// TIA Portal V17 export
// export: Created 2024-06-14T09:53:09.4288461Z, ExportSetting WithDefaults, DisplayName Totally Integrated Automation Portal, DisplayVersion V17, DisplayName TIA Portal Openness, DisplayVersion V17, DisplayName TIA Portal Version Control Interface, DisplayVersion V17, DisplayName Simotion SCOUT TIA, DisplayVersion 5.4.3.0, DisplayName SINAMICS Startdrive Advanced, DisplayVersion V17 SP1 Update 1, DisplayName SINAMICS Startdrive G110M, G120, G120C, G120D, G120P, G115D, DisplayVersion V17 SP1 Update 1, DisplayName SINAMICS Startdrive G130, G150, S120, S150, SINAMICS MV, S210, DisplayVersion V17 SP1 Update 1, DisplayName STEP 7 Professional, DisplayVersion V17, DisplayName STEP 7 Safety, DisplayVersion V17, DisplayName WinCC Professional, DisplayVersion V17
FUNCTION_BLOCK "LPG_Check_scale_FB"   // FB102, LAD
TITLE = Fiiling Operation FB
{ S7_Optimized_Access := 'TRUE' }
VERSION : 0.1
// stored: AutoNumber false, IsIECCheckEnabled false, IsRetainMemResEnabled false, MemoryReserve 100, SetENOAutomatically false, UDAEnableTagReadback false
   VAR_INPUT
      INxCylinder_In_Pos : Bool;   // Cylinder In Position
      INxAuto_Start_Seq : Bool;   // Start Filling Sequence
      INxMan_Start_Seq : Bool;
      INxStop_Sequence : Bool;   // Stop Filling Sequence
      INtStart_TImeout_Time : DInt;   // Start Timeout Time in Sec
      INxReset_Sequence : Bool;   // Reset Sequence
      INxCylinder_Type : Int;
      INrTare_Entry_SP : Real;
      DOWN_CONVEYOR : Bool;
      data_delete : Bool;
   END_VAR
   VAR_OUTPUT
      OutuFilled_Data : Array[1..10] of Real;
      OutxDomestic_Cylinder : Bool;
      OutxCommercial_Cylinder : Bool;
      OutxStart_Timeout : Bool;
      OutxTare_Entry_Error : Bool;   // Coil 27
      Outx_Filling_Error : Bool;
      Outx_Tare_Value_Error : Bool;
      Cycle_Started : Bool;
      OutiStep_No : Int;
      OUTiResult : Int;
      Gross_Weight : Real;
      Net_Wieght : Real;
      Tare_Weight : Real;
      OUT_Decision : Int;
   END_VAR
   VAR_IN_OUT
      Modbus_Master_DB : "MOD_MASTER_DATA_1";
   END_VAR
   VAR
      TRIG : Array[1..25] of Bool;
      STEP_NO : Int;
      Step_Timer { S7_SetPoint := 'True'} : Array[1..15] of IEC_TIMER;
      Domestic_Cylinder { S7_SetPoint := 'True'} : Bool;
      Commercial_Cylinder : Bool;
      Cyl_Done { S7_SetPoint := 'True'} : TOF_TIME;
      Tare_Enrty_Extn { S7_SetPoint := 'True'} : TOF_TIME;
      Start_Timeout_Err { S7_SetPoint := 'True'} : TON_TIME;
      Tare_Entry_Timer { S7_SetPoint := 'True'} : TON_TIME;
      Filled_Gross : Real;
      Filled_Net : Real;
      Punched_Tare : Real;
      Test_Seq : Int;
      RESULT : Bool;
      IEC_Timer_0_Instance { S7_SetPoint := 'True'} : TOF_TIME;
      Gross { S7_SetPoint := 'True'} : Real;
      gross_diff : Real;
      pass : Bool;
      Decision : Word;
      IEC_Timer_0_Instance_1 { S7_SetPoint := 'True'} : TON_TIME;
      fill { S7_SetPoint := 'True'} : TON_TIME;
      ALL_FILL_DONE : Bool;
   END_VAR
   VAR RETAIN
      cycle_start { S7_SetPoint := 'True'} : CTU_INT;
   END_VAR
   VAR_TEMP
      Tare_Weight_Mul : Real;
      Tare_Enter_Time : DInt;
      Stt_TImeout_Time : DInt;
      Tare_Entry_Time : DInt;
      Tare_SP_Weigher : Int;
      Filled_Gross_Mul : Int;
      Filled_Net_Mul : Int;
      Filled_Tare_Mul : Int;
      "final wieght" : Real;
      final_weight_1 : Real;
   END_VAR
   // Tare_Enrty_Extn.PT := T#1s;
   VAR_TEMP   // added for the SCL form of the ladder/FBD networks
      _w1 : Bool;
      _w2 : Bool;
      _w3 : Bool;
   END_VAR
BEGIN

REGION Network 1: Empty Network
END_REGION

REGION Network 2: Input Mapping
END_REGION

REGION Network 3: Cylinder Selection ( Domestic / Commercial )
   // We have to receive from FIFO Entry-
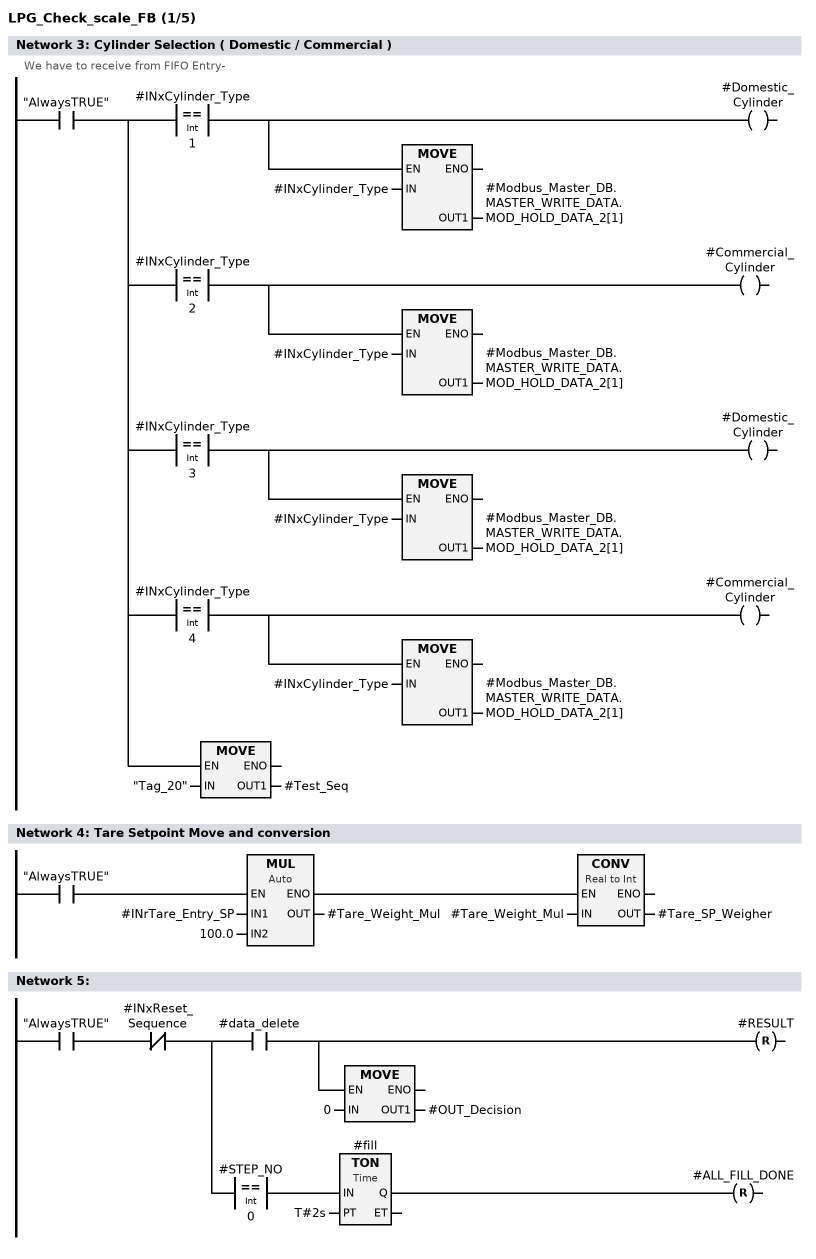
   RUNG wire#powerrail
      Contact( "AlwaysTRUE" )
      wire#w1
      { S7_Templates := "SrcType := Int" } EQ_Contact(in1 := #INxCylinder_Type, in2 := 1)
      wire#w2
      Coil( #Domestic_Cylinder )
   END_RUNG
   RUNG wire#w2
      Move(in := #INxCylinder_Type, out1 => #Modbus_Master_DB.MASTER_WRITE_DATA.MOD_HOLD_DATA_2[1])
   END_RUNG
   RUNG wire#w1
      { S7_Templates := "SrcType := Int" } EQ_Contact(in1 := #INxCylinder_Type, in2 := 2)
      wire#w3
      Coil( #Commercial_Cylinder )
   END_RUNG
   RUNG wire#w3
      Move(in := #INxCylinder_Type, out1 => #Modbus_Master_DB.MASTER_WRITE_DATA.MOD_HOLD_DATA_2[1])
   END_RUNG
   RUNG wire#w1
      { S7_Templates := "SrcType := Int" } EQ_Contact(in1 := #INxCylinder_Type, in2 := 3)
      wire#w4
      Coil( #Domestic_Cylinder )
   END_RUNG
   RUNG wire#w4
      Move(in := #INxCylinder_Type, out1 => #Modbus_Master_DB.MASTER_WRITE_DATA.MOD_HOLD_DATA_2[1])
   END_RUNG
   RUNG wire#w1
      { S7_Templates := "SrcType := Int" } EQ_Contact(in1 := #INxCylinder_Type, in2 := 4)
      wire#w5
      Coil( #Commercial_Cylinder )
   END_RUNG
   RUNG wire#w5
      Move(in := #INxCylinder_Type, out1 => #Modbus_Master_DB.MASTER_WRITE_DATA.MOD_HOLD_DATA_2[1])
   END_RUNG
   RUNG wire#w1
      Move(in := "Tag_20", out1 => #Test_Seq)
   END_RUNG
   // the same network as SCL:
   #Domestic_Cylinder := "AlwaysTRUE" AND (#INxCylinder_Type = 1);
   IF #Domestic_Cylinder THEN
       #Modbus_Master_DB.MASTER_WRITE_DATA.MOD_HOLD_DATA_2[1] := #INxCylinder_Type;
   END_IF;
   #Commercial_Cylinder := "AlwaysTRUE" AND (#INxCylinder_Type = 2);
   IF #Commercial_Cylinder THEN
       #Modbus_Master_DB.MASTER_WRITE_DATA.MOD_HOLD_DATA_2[1] := #INxCylinder_Type;
   END_IF;
   #Domestic_Cylinder := "AlwaysTRUE" AND (#INxCylinder_Type = 3);
   IF #Domestic_Cylinder THEN
       #Modbus_Master_DB.MASTER_WRITE_DATA.MOD_HOLD_DATA_2[1] := #INxCylinder_Type;
   END_IF;
   #Commercial_Cylinder := "AlwaysTRUE" AND (#INxCylinder_Type = 4);
   IF #Commercial_Cylinder THEN
       #Modbus_Master_DB.MASTER_WRITE_DATA.MOD_HOLD_DATA_2[1] := #INxCylinder_Type;
   END_IF;
   IF "AlwaysTRUE" THEN #Test_Seq := "Tag_20"; END_IF;
END_REGION

REGION Network 4: Tare Setpoint Move and conversion
   RUNG wire#powerrail
      Contact( "AlwaysTRUE" )
      Mul(in1 := #INrTare_Entry_SP, in2 := 100.0, out => #Tare_Weight_Mul)
      { S7_Templates := "[SrcType := Real, DestType := Int]" } Convert(in := #Tare_Weight_Mul, out => #Tare_SP_Weigher)
   END_RUNG
   // the same network as SCL:
   IF "AlwaysTRUE" THEN
       #Tare_Weight_Mul := #INrTare_Entry_SP * 100.0;
       #Tare_SP_Weigher := REAL_TO_INT(#Tare_Weight_Mul);
   END_IF;
END_REGION

REGION Network 5
   RUNG wire#powerrail
      Contact( "AlwaysTRUE" )
      I_Contact( #INxReset_Sequence )
      wire#w1
      Contact( #data_delete )
      wire#w2
      R_Coil( #RESULT )
   END_RUNG
   RUNG wire#w2
      Move(in := 0, out1 => #OUT_Decision)
   END_RUNG
   RUNG wire#w1
      { S7_Templates := "SrcType := Int" } EQ_Contact(in1 := #STEP_NO, in2 := 0)
      { S7_Templates := "time_type := Time" } #fill.TON(pt := T#2s, et =>)
      R_Coil( #ALL_FILL_DONE )
   END_RUNG
   // the same network as SCL:
   #_w1 := "AlwaysTRUE" AND NOT #INxReset_Sequence;
   IF #_w1 AND #data_delete THEN
       #RESULT := FALSE;
       #OUT_Decision := 0;
   END_IF;
   #fill(IN := #_w1 AND (#STEP_NO = 0), PT := T#2s);   // TON
   IF #fill.Q THEN #ALL_FILL_DONE := FALSE; END_IF;
END_REGION

REGION Network 6: Cylinder Selection
   // Cylinder Selection will write the logic later
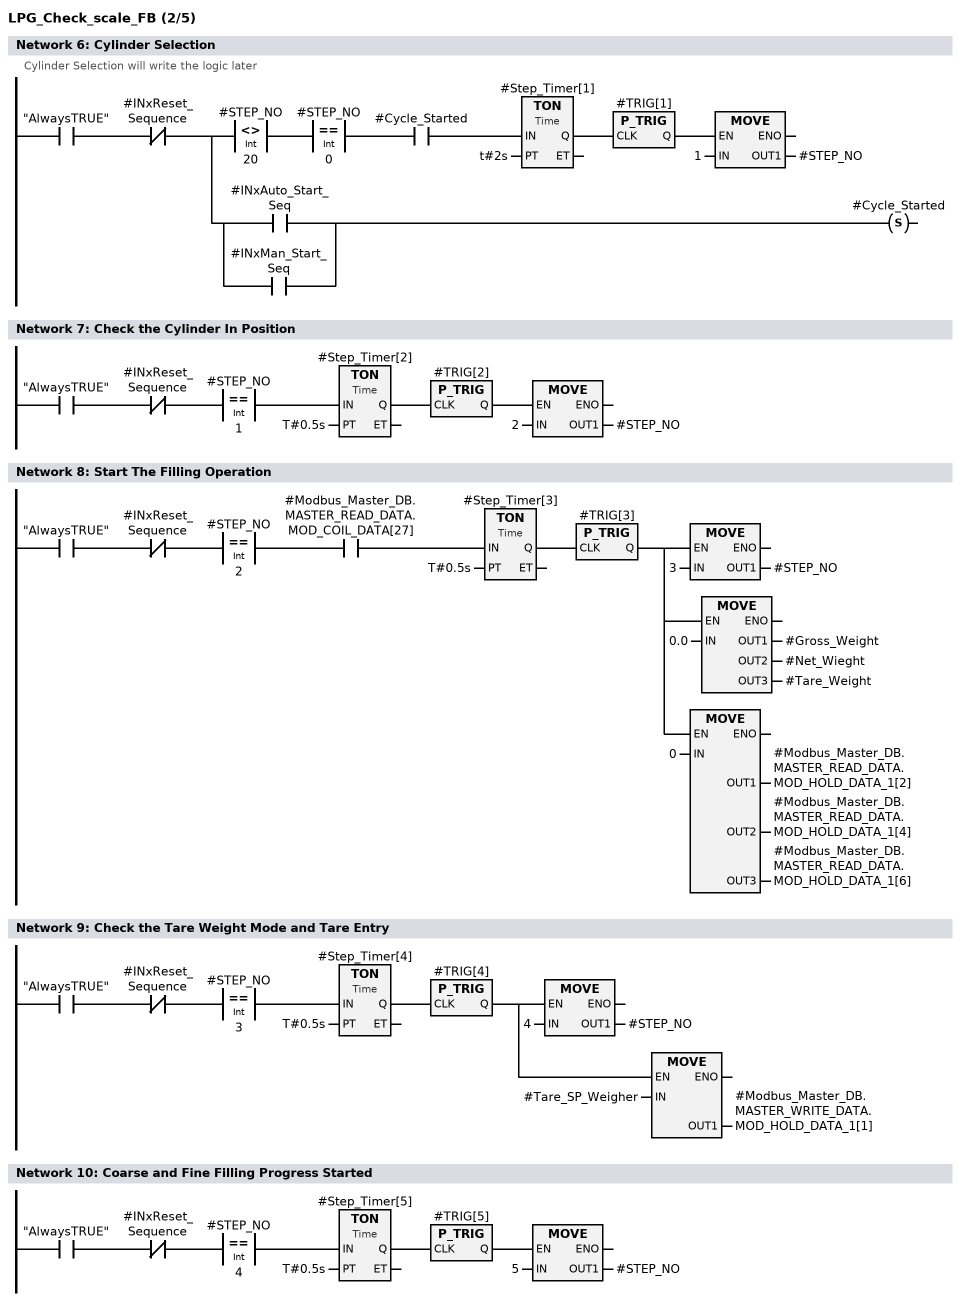
   RUNG wire#powerrail
      Contact( "AlwaysTRUE" )
      I_Contact( #INxReset_Sequence )
      wire#w1
      { S7_Templates := "SrcType := Int" } NE_Contact(in1 := #STEP_NO, in2 := 20)
      { S7_Templates := "SrcType := Int" } EQ_Contact(in1 := #STEP_NO, in2 := 0)
      Contact( #Cycle_Started )
      { S7_Templates := "time_type := Time" } #Step_Timer[1].TON(pt := t#2s, et =>)
      P_Trig( #TRIG[1] )
      Move(in := 1, out1 => #STEP_NO)
   END_RUNG
   RUNG wire#w1
      Contact( #INxAuto_Start_Seq )
      wire#w2
      S_Coil( #Cycle_Started )
   END_RUNG
   RUNG wire#w1
      Contact( #INxMan_Start_Seq )
   END_RUNG wire#w2
   // the same network as SCL:
   #_w1 := "AlwaysTRUE" AND NOT #INxReset_Sequence;
   #Step_Timer[1].TON(IN := #_w1 AND (#STEP_NO <> 20) AND (#STEP_NO = 0) AND #Cycle_Started, PT := t#2s);
   #_w2 := #Step_Timer[1].Q AND NOT #TRIG[1];   // rising edge
   #TRIG[1] := #Step_Timer[1].Q;
   IF #_w2 THEN #STEP_NO := 1; END_IF;
   IF #_w1 AND (#INxAuto_Start_Seq OR #INxMan_Start_Seq) THEN #Cycle_Started := TRUE; END_IF;
END_REGION

REGION Network 7: Check the Cylinder In Position
   RUNG wire#powerrail
      Contact( "AlwaysTRUE" )
      I_Contact( #INxReset_Sequence )
      { S7_Templates := "SrcType := Int" } EQ_Contact(in1 := #STEP_NO, in2 := 1)
      { S7_Templates := "time_type := Time" } #Step_Timer[2].TON(pt := T#0.5s, et =>)
      P_Trig( #TRIG[2] )
      Move(in := 2, out1 => #STEP_NO)
   END_RUNG
   // the same network as SCL:
   #Step_Timer[2].TON(IN := "AlwaysTRUE" AND NOT #INxReset_Sequence AND (#STEP_NO = 1), PT := T#0.5s);
   #_w1 := #Step_Timer[2].Q AND NOT #TRIG[2];   // rising edge
   #TRIG[2] := #Step_Timer[2].Q;
   IF #_w1 THEN #STEP_NO := 2; END_IF;
END_REGION

REGION Network 8: Start The Filling Operation
   RUNG wire#powerrail
      Contact( "AlwaysTRUE" )
      I_Contact( #INxReset_Sequence )
      { S7_Templates := "SrcType := Int" } EQ_Contact(in1 := #STEP_NO, in2 := 2)
      Contact( #Modbus_Master_DB.MASTER_READ_DATA.MOD_COIL_DATA[27] )
      { S7_Templates := "time_type := Time" } #Step_Timer[3].TON(pt := T#0.5s, et =>)
      P_Trig( #TRIG[3] )
      wire#w1
      Move(in := 3, out1 => #STEP_NO)
   END_RUNG
   RUNG wire#w1
      Move(in := 0.0, out1 => #Gross_Weight, out2 => #Net_Wieght, out3 => #Tare_Weight)
   END_RUNG
   RUNG wire#w1
      Move(in := 0, out1 => #Modbus_Master_DB.MASTER_READ_DATA.MOD_HOLD_DATA_1[2], out2 => #Modbus_Master_DB.MASTER_READ_DATA.MOD_HOLD_DATA_1[4], out3 => #Modbus_Master_DB.MASTER_READ_DATA.MOD_HOLD_DATA_1[6])
   END_RUNG
   // the same network as SCL:
   #Step_Timer[3].TON(IN := "AlwaysTRUE" AND NOT #INxReset_Sequence AND (#STEP_NO = 2) AND #Modbus_Master_DB.MASTER_READ_DATA.MOD_COIL_DATA[27],
                      PT := T#0.5s);
   #_w1 := #Step_Timer[3].Q AND NOT #TRIG[3];   // rising edge
   #TRIG[3] := #Step_Timer[3].Q;
   IF #_w1 THEN
       #STEP_NO := 3;
       #Gross_Weight := 0.0;
       #Net_Wieght := 0.0;
       #Tare_Weight := 0.0;
       #Modbus_Master_DB.MASTER_READ_DATA.MOD_HOLD_DATA_1[2] := 0;
       #Modbus_Master_DB.MASTER_READ_DATA.MOD_HOLD_DATA_1[4] := 0;
       #Modbus_Master_DB.MASTER_READ_DATA.MOD_HOLD_DATA_1[6] := 0;
   END_IF;
END_REGION

REGION Network 9: Check the Tare Weight Mode and Tare Entry
   RUNG wire#powerrail
      Contact( "AlwaysTRUE" )
      I_Contact( #INxReset_Sequence )
      { S7_Templates := "SrcType := Int" } EQ_Contact(in1 := #STEP_NO, in2 := 3)
      { S7_Templates := "time_type := Time" } #Step_Timer[4].TON(pt := T#0.5s, et =>)
      P_Trig( #TRIG[4] )
      wire#w1
      Move(in := 4, out1 => #STEP_NO)
   END_RUNG
   RUNG wire#w1
      Move(in := #Tare_SP_Weigher, out1 => #Modbus_Master_DB.MASTER_WRITE_DATA.MOD_HOLD_DATA_1[1])
   END_RUNG
   // the same network as SCL:
   #Step_Timer[4].TON(IN := "AlwaysTRUE" AND NOT #INxReset_Sequence AND (#STEP_NO = 3), PT := T#0.5s);
   #_w1 := #Step_Timer[4].Q AND NOT #TRIG[4];   // rising edge
   #TRIG[4] := #Step_Timer[4].Q;
   IF #_w1 THEN
       #STEP_NO := 4;
       #Modbus_Master_DB.MASTER_WRITE_DATA.MOD_HOLD_DATA_1[1] := #Tare_SP_Weigher;
   END_IF;
END_REGION

REGION Network 10: Coarse and Fine Filling Progress Started
   RUNG wire#powerrail
      Contact( "AlwaysTRUE" )
      I_Contact( #INxReset_Sequence )
      { S7_Templates := "SrcType := Int" } EQ_Contact(in1 := #STEP_NO, in2 := 4)
      { S7_Templates := "time_type := Time" } #Step_Timer[5].TON(pt := T#0.5s, et =>)
      P_Trig( #TRIG[5] )
      Move(in := 5, out1 => #STEP_NO)
   END_RUNG
   // the same network as SCL:
   #Step_Timer[5].TON(IN := "AlwaysTRUE" AND NOT #INxReset_Sequence AND (#STEP_NO = 4), PT := T#0.5s);
   #_w1 := #Step_Timer[5].Q AND NOT #TRIG[5];   // rising edge
   #TRIG[5] := #Step_Timer[5].Q;
   IF #_w1 THEN #STEP_NO := 5; END_IF;
END_REGION

REGION Network 11: Coarse Filling Completed
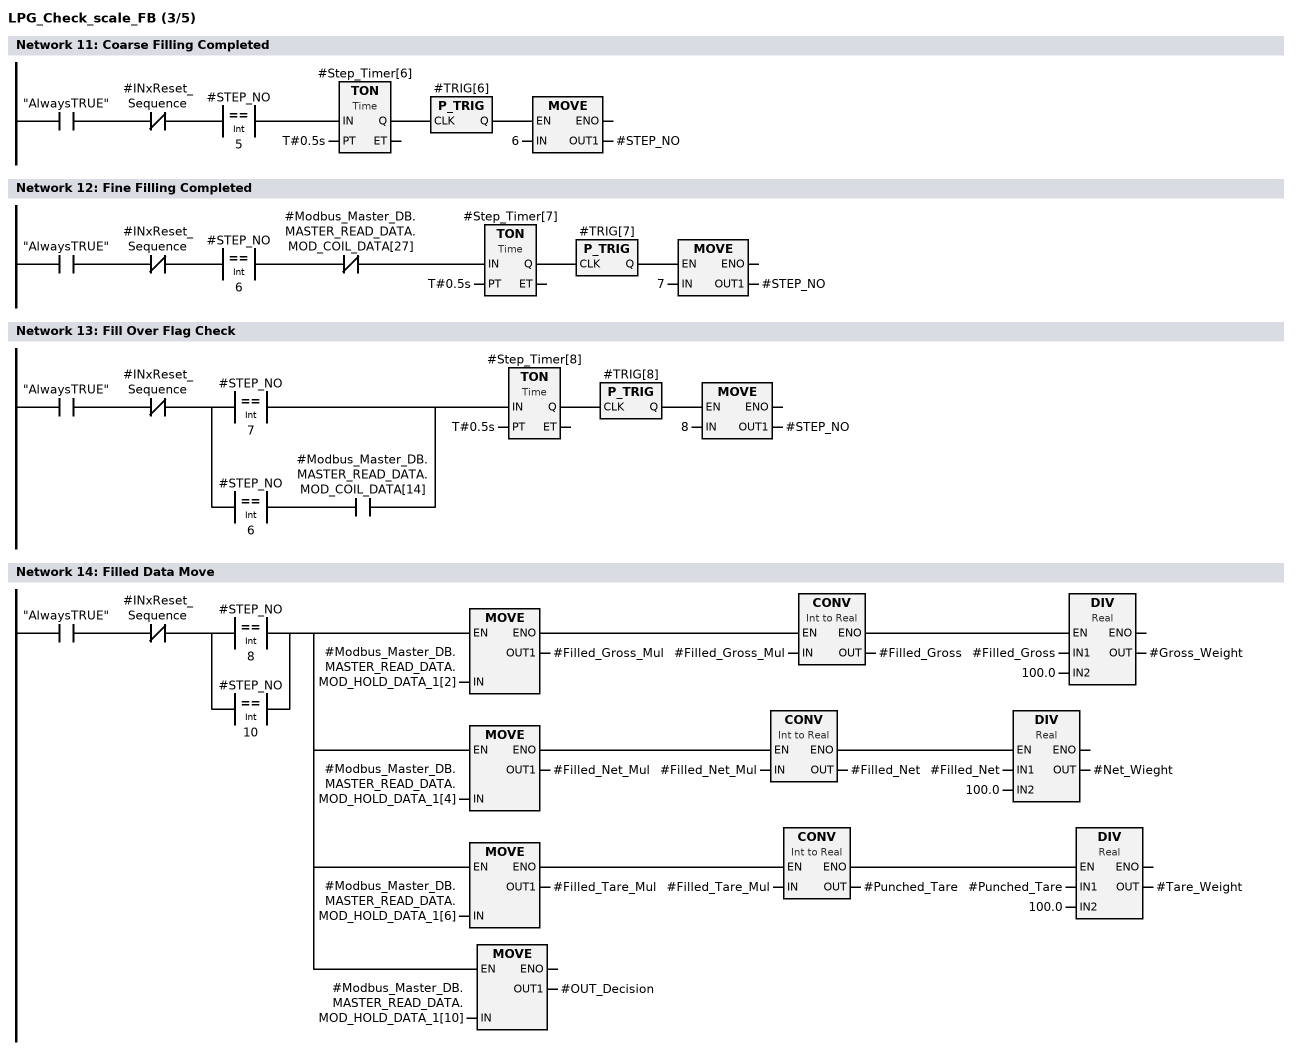
   RUNG wire#powerrail
      Contact( "AlwaysTRUE" )
      I_Contact( #INxReset_Sequence )
      { S7_Templates := "SrcType := Int" } EQ_Contact(in1 := #STEP_NO, in2 := 5)
      { S7_Templates := "time_type := Time" } #Step_Timer[6].TON(pt := T#0.5s, et =>)
      P_Trig( #TRIG[6] )
      Move(in := 6, out1 => #STEP_NO)
   END_RUNG
   // the same network as SCL:
   #Step_Timer[6].TON(IN := "AlwaysTRUE" AND NOT #INxReset_Sequence AND (#STEP_NO = 5), PT := T#0.5s);
   #_w1 := #Step_Timer[6].Q AND NOT #TRIG[6];   // rising edge
   #TRIG[6] := #Step_Timer[6].Q;
   IF #_w1 THEN #STEP_NO := 6; END_IF;
END_REGION

REGION Network 12: Fine Filling Completed
   RUNG wire#powerrail
      Contact( "AlwaysTRUE" )
      I_Contact( #INxReset_Sequence )
      { S7_Templates := "SrcType := Int" } EQ_Contact(in1 := #STEP_NO, in2 := 6)
      I_Contact( #Modbus_Master_DB.MASTER_READ_DATA.MOD_COIL_DATA[27] )
      { S7_Templates := "time_type := Time" } #Step_Timer[7].TON(pt := T#0.5s, et =>)
      P_Trig( #TRIG[7] )
      Move(in := 7, out1 => #STEP_NO)
   END_RUNG
   // the same network as SCL:
   #Step_Timer[7].TON(IN := "AlwaysTRUE" AND NOT #INxReset_Sequence AND (#STEP_NO = 6) AND NOT #Modbus_Master_DB.MASTER_READ_DATA.MOD_COIL_DATA[27],
                      PT := T#0.5s);
   #_w1 := #Step_Timer[7].Q AND NOT #TRIG[7];   // rising edge
   #TRIG[7] := #Step_Timer[7].Q;
   IF #_w1 THEN #STEP_NO := 7; END_IF;
END_REGION

REGION Network 13: Fill Over Flag Check
   RUNG wire#powerrail
      Contact( "AlwaysTRUE" )
      I_Contact( #INxReset_Sequence )
      wire#w1
      { S7_Templates := "SrcType := Int" } EQ_Contact(in1 := #STEP_NO, in2 := 7)
      wire#w2
      { S7_Templates := "time_type := Time" } #Step_Timer[8].TON(pt := T#0.5s, et =>)
      P_Trig( #TRIG[8] )
      Move(in := 8, out1 => #STEP_NO)
   END_RUNG
   RUNG wire#w1
      { S7_Templates := "SrcType := Int" } EQ_Contact(in1 := #STEP_NO, in2 := 6)
      Contact( #Modbus_Master_DB.MASTER_READ_DATA.MOD_COIL_DATA[14] )
   END_RUNG wire#w2
   // the same network as SCL:
   #Step_Timer[8].TON(IN := "AlwaysTRUE" AND NOT #INxReset_Sequence AND ((#STEP_NO = 7) OR ((#STEP_NO = 6) AND #Modbus_Master_DB.MASTER_READ_DATA.MOD_COIL_DATA[14])),
                      PT := T#0.5s);
   #_w1 := #Step_Timer[8].Q AND NOT #TRIG[8];   // rising edge
   #TRIG[8] := #Step_Timer[8].Q;
   IF #_w1 THEN #STEP_NO := 8; END_IF;
END_REGION

REGION Network 14: Filled Data Move
   RUNG wire#powerrail
      Contact( "AlwaysTRUE" )
      I_Contact( #INxReset_Sequence )
      wire#w1
      { S7_Templates := "SrcType := Int" } EQ_Contact(in1 := #STEP_NO, in2 := 8)
      wire#w2
      Move(in := #Modbus_Master_DB.MASTER_READ_DATA.MOD_HOLD_DATA_1[2], out1 => #Filled_Gross_Mul)
      { S7_Templates := "[SrcType := Int, DestType := Real]" } Convert(in := #Filled_Gross_Mul, out => #Filled_Gross)
      { S7_Templates := "SrcType := Real" } Div(in1 := #Filled_Gross, in2 := 100.0, out => #Gross_Weight)
   END_RUNG
   RUNG wire#w1
      { S7_Templates := "SrcType := Int" } EQ_Contact(in1 := #STEP_NO, in2 := 10)
   END_RUNG wire#w2
   RUNG wire#w2
      Move(in := #Modbus_Master_DB.MASTER_READ_DATA.MOD_HOLD_DATA_1[4], out1 => #Filled_Net_Mul)
      { S7_Templates := "[SrcType := Int, DestType := Real]" } Convert(in := #Filled_Net_Mul, out => #Filled_Net)
      { S7_Templates := "SrcType := Real" } Div(in1 := #Filled_Net, in2 := 100.0, out => #Net_Wieght)
   END_RUNG
   RUNG wire#w2
      Move(in := #Modbus_Master_DB.MASTER_READ_DATA.MOD_HOLD_DATA_1[6], out1 => #Filled_Tare_Mul)
      { S7_Templates := "[SrcType := Int, DestType := Real]" } Convert(in := #Filled_Tare_Mul, out => #Punched_Tare)
      { S7_Templates := "SrcType := Real" } Div(in1 := #Punched_Tare, in2 := 100.0, out => #Tare_Weight)
   END_RUNG
   RUNG wire#w2
      Move(in := #Modbus_Master_DB.MASTER_READ_DATA.MOD_HOLD_DATA_1[10], out1 => #OUT_Decision)
   END_RUNG
   // the same network as SCL:
   IF "AlwaysTRUE" AND NOT #INxReset_Sequence AND ((#STEP_NO = 8) OR (#STEP_NO = 10)) THEN
       #Filled_Gross_Mul := #Modbus_Master_DB.MASTER_READ_DATA.MOD_HOLD_DATA_1[2];
       #Filled_Gross := INT_TO_REAL(#Filled_Gross_Mul);
       #Gross_Weight := #Filled_Gross / 100.0;
       #Filled_Net_Mul := #Modbus_Master_DB.MASTER_READ_DATA.MOD_HOLD_DATA_1[4];
       #Filled_Net := INT_TO_REAL(#Filled_Net_Mul);
       #Net_Wieght := #Filled_Net / 100.0;
       #Filled_Tare_Mul := #Modbus_Master_DB.MASTER_READ_DATA.MOD_HOLD_DATA_1[6];
       #Punched_Tare := INT_TO_REAL(#Filled_Tare_Mul);
       #Tare_Weight := #Punched_Tare / 100.0;
       #OUT_Decision := #Modbus_Master_DB.MASTER_READ_DATA.MOD_HOLD_DATA_1[10];
   END_IF;
END_REGION

REGION Network 15: Filling Operation Complete
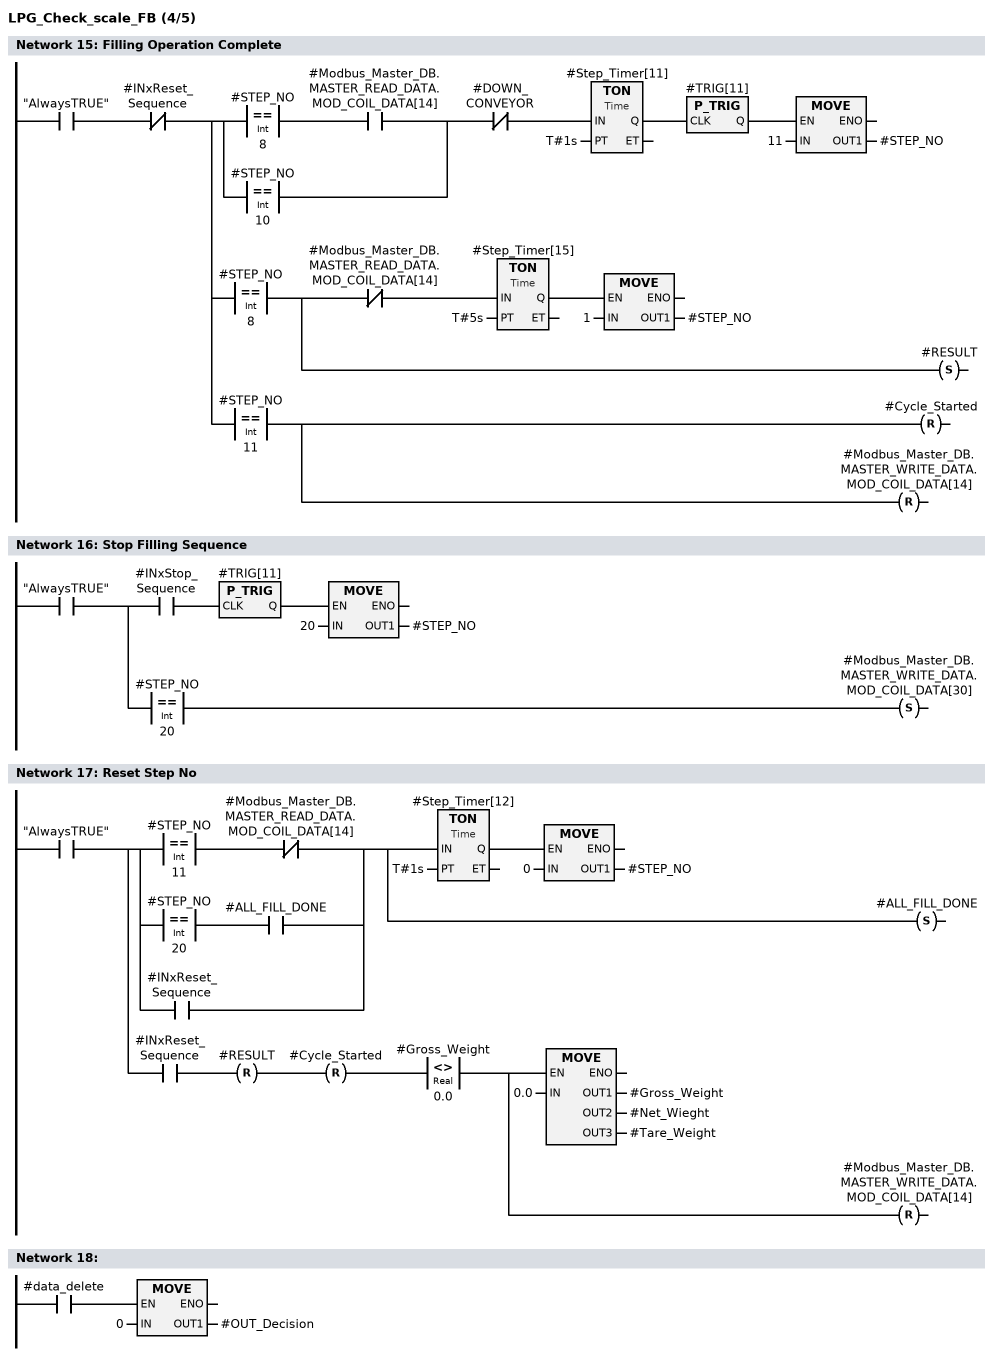
   RUNG wire#powerrail
      Contact( "AlwaysTRUE" )
      I_Contact( #INxReset_Sequence )
      wire#w1
      { S7_Templates := "SrcType := Int" } EQ_Contact(in1 := #STEP_NO, in2 := 8)
      Contact( #Modbus_Master_DB.MASTER_READ_DATA.MOD_COIL_DATA[14] )
      wire#w2
      I_Contact( #DOWN_CONVEYOR )
      { S7_Templates := "time_type := Time" } #Step_Timer[11].TON(pt := T#1s, et =>)
      P_Trig( #TRIG[11] )
      Move(in := 11, out1 => #STEP_NO)
   END_RUNG
   RUNG wire#w1
      { S7_Templates := "SrcType := Int" } EQ_Contact(in1 := #STEP_NO, in2 := 10)
   END_RUNG wire#w2
   RUNG wire#w1
      { S7_Templates := "SrcType := Int" } EQ_Contact(in1 := #STEP_NO, in2 := 8)
      wire#w3
      I_Contact( #Modbus_Master_DB.MASTER_READ_DATA.MOD_COIL_DATA[14] )
      { S7_Templates := "time_type := Time" } #Step_Timer[15].TON(pt := T#5s, et =>)
      Move(in := 1, out1 => #STEP_NO)
   END_RUNG
   RUNG wire#w3
      S_Coil( #RESULT )
   END_RUNG
   RUNG wire#w1
      { S7_Templates := "SrcType := Int" } EQ_Contact(in1 := #STEP_NO, in2 := 11)
      wire#w4
      R_Coil( #Cycle_Started )
   END_RUNG
   RUNG wire#w4
      R_Coil( #Modbus_Master_DB.MASTER_WRITE_DATA.MOD_COIL_DATA[14] )
   END_RUNG
   // the same network as SCL:
   #_w1 := "AlwaysTRUE" AND NOT #INxReset_Sequence;
   #Step_Timer[11].TON(IN := #_w1 AND (((#STEP_NO = 8) AND #Modbus_Master_DB.MASTER_READ_DATA.MOD_COIL_DATA[14]) OR (#STEP_NO = 10)) AND NOT #DOWN_CONVEYOR,
                       PT := T#1s);
   #_w2 := #Step_Timer[11].Q AND NOT #TRIG[11];   // rising edge
   #TRIG[11] := #Step_Timer[11].Q;
   IF #_w2 THEN #STEP_NO := 11; END_IF;
   #_w3 := #_w1 AND (#STEP_NO = 8);
   #Step_Timer[15].TON(IN := #_w3 AND NOT #Modbus_Master_DB.MASTER_READ_DATA.MOD_COIL_DATA[14], PT := T#5s);
   IF #Step_Timer[15].Q THEN #STEP_NO := 1; END_IF;
   IF #_w3 THEN #RESULT := TRUE; END_IF;
   IF #_w1 AND (#STEP_NO = 11) THEN
       #Cycle_Started := FALSE;
       #Modbus_Master_DB.MASTER_WRITE_DATA.MOD_COIL_DATA[14] := FALSE;
   END_IF;
END_REGION

REGION Network 16: Stop Filling Sequence
   RUNG wire#powerrail
      Contact( "AlwaysTRUE" )
      wire#w1
      Contact( #INxStop_Sequence )
      P_Trig( #TRIG[11] )
      Move(in := 20, out1 => #STEP_NO)
   END_RUNG
   RUNG wire#w1
      { S7_Templates := "SrcType := Int" } EQ_Contact(in1 := #STEP_NO, in2 := 20)
      S_Coil( #Modbus_Master_DB.MASTER_WRITE_DATA.MOD_COIL_DATA[30] )
   END_RUNG
   // the same network as SCL:
   #_w1 := "AlwaysTRUE" AND #INxStop_Sequence;
   #_w2 := #_w1 AND NOT #TRIG[11];   // rising edge
   #TRIG[11] := #_w1;
   IF #_w2 THEN #STEP_NO := 20; END_IF;
   IF "AlwaysTRUE" AND (#STEP_NO = 20) THEN
       #Modbus_Master_DB.MASTER_WRITE_DATA.MOD_COIL_DATA[30] := TRUE;
   END_IF;
END_REGION

REGION Network 17: Reset Step No
   RUNG wire#powerrail
      Contact( "AlwaysTRUE" )
      wire#w1
      { S7_Templates := "SrcType := Int" } EQ_Contact(in1 := #STEP_NO, in2 := 11)
      I_Contact( #Modbus_Master_DB.MASTER_READ_DATA.MOD_COIL_DATA[14] )
      wire#w2
      { S7_Templates := "time_type := Time" } #Step_Timer[12].TON(pt := T#1s, et =>)
      Move(in := 0, out1 => #STEP_NO)
   END_RUNG
   RUNG wire#w1
      { S7_Templates := "SrcType := Int" } EQ_Contact(in1 := #STEP_NO, in2 := 20)
      Contact( #ALL_FILL_DONE )
   END_RUNG wire#w2
   RUNG wire#w1
      Contact( #INxReset_Sequence )
   END_RUNG wire#w2
   RUNG wire#w2
      S_Coil( #ALL_FILL_DONE )
   END_RUNG
   RUNG wire#w1
      Contact( #INxReset_Sequence )
      R_Coil( #RESULT )
      R_Coil( #Cycle_Started )
      { S7_Templates := "SrcType := Real" } NE_Contact(in1 := #Gross_Weight, in2 := 0.0)
      wire#w3
      Move(in := 0.0, out1 => #Gross_Weight, out2 => #Net_Wieght, out3 => #Tare_Weight)
   END_RUNG
   RUNG wire#w3
      R_Coil( #Modbus_Master_DB.MASTER_WRITE_DATA.MOD_COIL_DATA[14] )
   END_RUNG
   // the same network as SCL:
   #_w1 := "AlwaysTRUE" AND (((#STEP_NO = 11) AND NOT #Modbus_Master_DB.MASTER_READ_DATA.MOD_COIL_DATA[14]) OR ((#STEP_NO = 20) AND #ALL_FILL_DONE) OR #INxReset_Sequence);
   #Step_Timer[12].TON(IN := #_w1, PT := T#1s);
   IF #Step_Timer[12].Q THEN #STEP_NO := 0; END_IF;
   IF #_w1 THEN #ALL_FILL_DONE := TRUE; END_IF;
   #_w2 := "AlwaysTRUE" AND #INxReset_Sequence;
   IF #_w2 THEN
       #RESULT := FALSE;
       #Cycle_Started := FALSE;
   END_IF;
   #_w3 := #_w2 AND (#Gross_Weight <> 0.0);
   IF #_w3 THEN
       #Gross_Weight := 0.0;
       #Net_Wieght := 0.0;
       #Tare_Weight := 0.0;
       #Modbus_Master_DB.MASTER_WRITE_DATA.MOD_COIL_DATA[14] := FALSE;
   END_IF;
END_REGION

REGION Network 18
   RUNG wire#powerrail
      Contact( #data_delete )
      Move(in := 0, out1 => #OUT_Decision)
   END_RUNG
   // the same network as SCL:
   IF #data_delete THEN #OUT_Decision := 0; END_IF;
END_REGION

REGION Network 19: Output Mapping
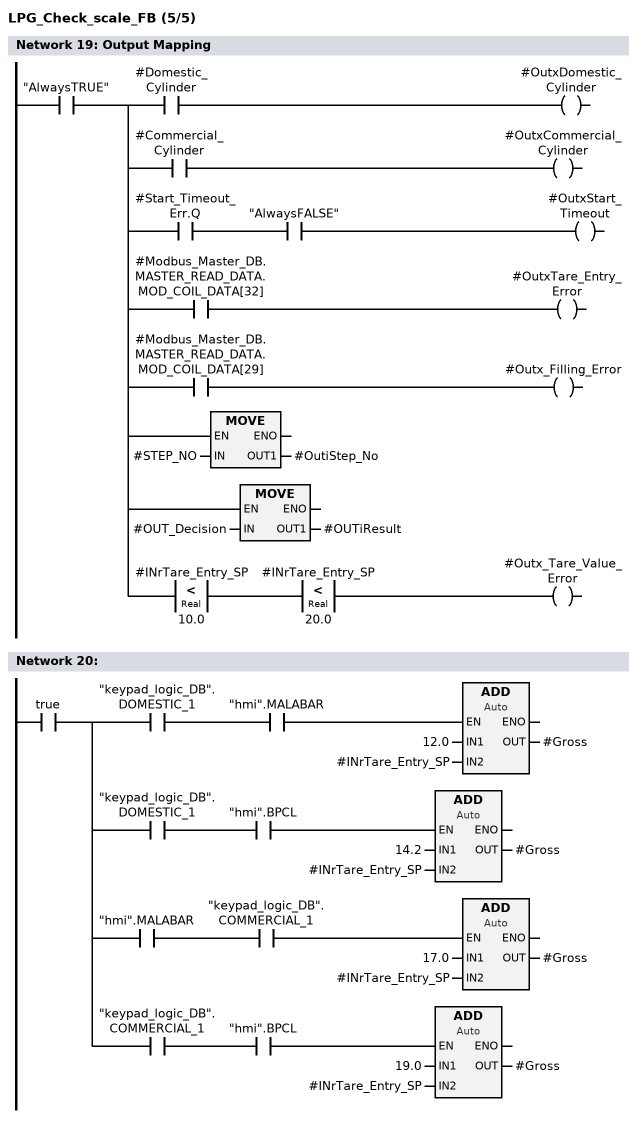
   RUNG wire#powerrail
      Contact( "AlwaysTRUE" )
      wire#w1
      Contact( #Domestic_Cylinder )
      Coil( #OutxDomestic_Cylinder )
   END_RUNG
   RUNG wire#w1
      Contact( #Commercial_Cylinder )
      Coil( #OutxCommercial_Cylinder )
   END_RUNG
   RUNG wire#w1
      Contact( #Start_Timeout_Err.Q )
      Contact( "AlwaysFALSE" )
      Coil( #OutxStart_Timeout )
   END_RUNG
   RUNG wire#w1
      Contact( #Modbus_Master_DB.MASTER_READ_DATA.MOD_COIL_DATA[32] )
      Coil( #OutxTare_Entry_Error )
   END_RUNG
   RUNG wire#w1
      Contact( #Modbus_Master_DB.MASTER_READ_DATA.MOD_COIL_DATA[29] )
      Coil( #Outx_Filling_Error )
   END_RUNG
   RUNG wire#w1
      Move(in := #STEP_NO, out1 => #OutiStep_No)
   END_RUNG
   RUNG wire#w1
      Move(in := #OUT_Decision, out1 => #OUTiResult)
   END_RUNG
   RUNG wire#w1
      { S7_Templates := "SrcType := Real" } LT_Contact(in1 := #INrTare_Entry_SP, in2 := 10.0)
      { S7_Templates := "SrcType := Real" } LT_Contact(in1 := #INrTare_Entry_SP, in2 := 20.0)
      Coil( #Outx_Tare_Value_Error )
   END_RUNG
   // the same network as SCL:
   #OutxDomestic_Cylinder := "AlwaysTRUE" AND #Domestic_Cylinder;
   #OutxCommercial_Cylinder := "AlwaysTRUE" AND #Commercial_Cylinder;
   #OutxStart_Timeout := "AlwaysTRUE" AND #Start_Timeout_Err.Q AND "AlwaysFALSE";
   #OutxTare_Entry_Error := "AlwaysTRUE" AND #Modbus_Master_DB.MASTER_READ_DATA.MOD_COIL_DATA[32];
   #Outx_Filling_Error := "AlwaysTRUE" AND #Modbus_Master_DB.MASTER_READ_DATA.MOD_COIL_DATA[29];
   IF "AlwaysTRUE" THEN
       #OutiStep_No := #STEP_NO;
       #OUTiResult := #OUT_Decision;
   END_IF;
   #Outx_Tare_Value_Error := "AlwaysTRUE" AND (#INrTare_Entry_SP < 10.0) AND (#INrTare_Entry_SP < 20.0);
END_REGION

REGION Network 20
   RUNG wire#powerrail
      Contact( true )
      wire#w1
      Contact( "keypad_logic_DB".DOMESTIC_1 )
      Contact( "hmi".MALABAR )
      Add(in1 := 12.0, in2 := #INrTare_Entry_SP, out => #Gross)
   END_RUNG
   RUNG wire#w1
      Contact( "keypad_logic_DB".DOMESTIC_1 )
      Contact( "hmi".BPCL )
      Add(in1 := 14.2, in2 := #INrTare_Entry_SP, out => #Gross)
   END_RUNG
   RUNG wire#w1
      Contact( "hmi".MALABAR )
      Contact( "keypad_logic_DB".COMMERCIAL_1 )
      Add(in1 := 17.0, in2 := #INrTare_Entry_SP, out => #Gross)
   END_RUNG
   RUNG wire#w1
      Contact( "keypad_logic_DB".COMMERCIAL_1 )
      Contact( "hmi".BPCL )
      Add(in1 := 19.0, in2 := #INrTare_Entry_SP, out => #Gross)
   END_RUNG
   // the same network as SCL:
   IF true AND "keypad_logic_DB".DOMESTIC_1 AND "hmi".MALABAR THEN
       #Gross := 12.0 + #INrTare_Entry_SP;
   END_IF;
   IF true AND "keypad_logic_DB".DOMESTIC_1 AND "hmi".BPCL THEN #Gross := 14.2 + #INrTare_Entry_SP; END_IF;
   IF true AND "hmi".MALABAR AND "keypad_logic_DB".COMMERCIAL_1 THEN
       #Gross := 17.0 + #INrTare_Entry_SP;
   END_IF;
   IF true AND "keypad_logic_DB".COMMERCIAL_1 AND "hmi".BPCL THEN #Gross := 19.0 + #INrTare_Entry_SP; END_IF;
END_REGION
END_FUNCTION_BLOCK
